TYPE TL_BUSY :
(
	eTlStartUnits := 0,
	eTlCheckUnits,
	eTlSignalError
)UINT;
END_TYPE

(* stored: Version 1.1.0.1, ProductVersion 3.1.4024.2
   DUT TL_BUSY: Id {34e15197-8fe8-4b82-9d95-d08600f63225} *)
